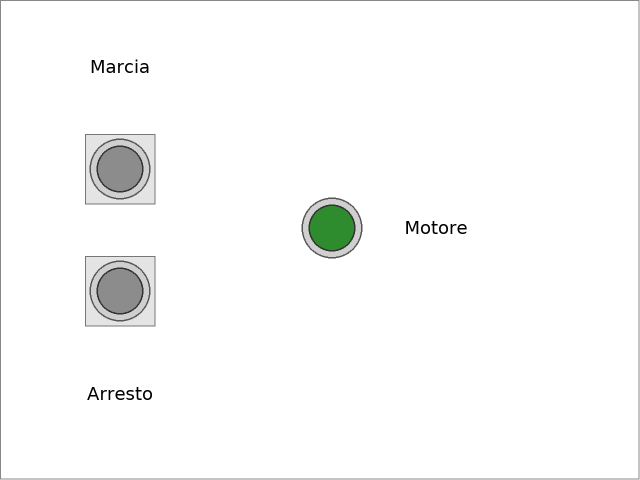
VISUALIZATION Screen1  // 640x480
    PushSwitch (85,134 70x70), variable: GVL.AvvioMotore, behaviour: TAP, style: Switch-PushSwitch-Gray
    PushSwitch (85,256 70x70), variable: GVL.ArrestoMotore, behaviour: TAP, style: Switch-PushSwitch-Gray
    Lamp1 (297,193 70x70), variable: GVL.MotoreInMarcia, style: Lamp-Lamp1-Green
    Label (361,213 150x30), "Motore"
    Label (45,52 150x30), "Marcia"
    Label (45,379 150x30), "Arresto"
END_VISUALIZATION

(* stored: Version 1.1.0.1, ProductVersion 3.1.4024.12
   Visu Screen1: Id {9b0049a9-98bb-4a53-a5c8-9865ebb9cb4b} *)
